// TIA Portal V18 export
DATA_BLOCK "DB 333"   // DB333
{ S7_Optimized_Access := 'FALSE' }
AUTHOR : AWP_S7P
FAMILY : WEB
VERSION : 1.0
// stored: AutoNumber false, DBAccessibleFromOPCUA true, IsOnlyStoredInLoadMemory false, IsWriteProtectedInAS false
   VAR
      magic { ExternalAccessible := 'False'; ExternalVisible := 'False'; ExternalWritable := 'False'} : DWord := DW#16#41575043;
      consistency_tag { ExternalAccessible := 'False'; ExternalVisible := 'False'; ExternalWritable := 'False'} : DWord := DW#16#0F12B01D;
      db_version { ExternalAccessible := 'False'; ExternalVisible := 'False'; ExternalWritable := 'False'} : Word := W#16#0001;
      length { ExternalAccessible := 'False'; ExternalVisible := 'False'; ExternalWritable := 'False'} : UInt := 586;
      pagetab_of { ExternalAccessible := 'False'; ExternalVisible := 'False'; ExternalWritable := 'False'} : UInt := 92;
      pagetab_count { ExternalAccessible := 'False'; ExternalVisible := 'False'; ExternalWritable := 'False'} : UInt := 4;
      excludetab_of { ExternalAccessible := 'False'; ExternalVisible := 'False'; ExternalWritable := 'False'} : UInt := 132;
      excludetab_count { ExternalAccessible := 'False'; ExternalVisible := 'False'; ExternalWritable := 'False'} : UInt := 0;
      fragmentlist_of { ExternalAccessible := 'False'; ExternalVisible := 'False'; ExternalWritable := 'False'} : UInt := 132;
      fragmentlist_count { ExternalAccessible := 'False'; ExternalVisible := 'False'; ExternalWritable := 'False'} : UInt := 5;
      fragmenttab_of { ExternalAccessible := 'False'; ExternalVisible := 'False'; ExternalWritable := 'False'} : UInt := 148;
      fragmenttab_count { ExternalAccessible := 'False'; ExternalVisible := 'False'; ExternalWritable := 'False'} : UInt := 5;
      datatab_of { ExternalAccessible := 'False'; ExternalVisible := 'False'; ExternalWritable := 'False'} : UInt := 218;
      datatab_count { ExternalAccessible := 'False'; ExternalVisible := 'False'; ExternalWritable := 'False'} : UInt := 2;
      usenametab_of { ExternalAccessible := 'False'; ExternalVisible := 'False'; ExternalWritable := 'False'} : UInt := 226;
      usenametab_count { ExternalAccessible := 'False'; ExternalVisible := 'False'; ExternalWritable := 'False'} : UInt := 0;
      enumreftab_of { ExternalAccessible := 'False'; ExternalVisible := 'False'; ExternalWritable := 'False'} : UInt := 226;
      enumreftab_count { ExternalAccessible := 'False'; ExternalVisible := 'False'; ExternalWritable := 'False'} : UInt := 0;
      enumtab_of { ExternalAccessible := 'False'; ExternalVisible := 'False'; ExternalWritable := 'False'} : UInt := 226;
      enumtab_count { ExternalAccessible := 'False'; ExternalVisible := 'False'; ExternalWritable := 'False'} : UInt := 0;
      textlist_of { ExternalAccessible := 'False'; ExternalVisible := 'False'; ExternalWritable := 'False'} : UInt := 226;
      textlist_count { ExternalAccessible := 'False'; ExternalVisible := 'False'; ExternalWritable := 'False'} : UInt := 360;
      language_frag_tab_of { ExternalAccessible := 'False'; ExternalVisible := 'False'; ExternalWritable := 'False'} : UInt := 142;
      language_frag_tab_count { ExternalAccessible := 'False'; ExternalVisible := 'False'; ExternalWritable := 'False'} : UInt := 6;
      application_name { ExternalAccessible := 'False'; ExternalVisible := 'False'; ExternalWritable := 'False'} : UInt := 1;
      application_url { ExternalAccessible := 'False'; ExternalVisible := 'False'; ExternalWritable := 'False'} : UInt := 19;
      application_desc { ExternalAccessible := 'False'; ExternalVisible := 'False'; ExternalWritable := 'False'} : UInt := 29;
      enum_defs_fragment_start { ExternalAccessible := 'False'; ExternalVisible := 'False'; ExternalWritable := 'False'} : UInt := 0;
      enum_defs_fragment_count { ExternalAccessible := 'False'; ExternalVisible := 'False'; ExternalWritable := 'False'} : UInt := 0;
      commandstate { ExternalAccessible := 'False'; ExternalVisible := 'False'; ExternalWritable := 'False'} : Struct
         last_error { ExternalAccessible := 'False'; ExternalVisible := 'False'; ExternalWritable := 'False'} : Int := 0;
         debug_mode { ExternalAccessible := 'False'; ExternalVisible := 'False'; ExternalWritable := 'False'} : Int := 0;
         init { ExternalAccessible := 'False'; ExternalVisible := 'False'; ExternalWritable := 'False'} : Bool := True;
         deactivate { ExternalAccessible := 'False'; ExternalVisible := 'False'; ExternalWritable := 'False'} : Bool := False;
         initializing { ExternalAccessible := 'False'; ExternalVisible := 'False'; ExternalWritable := 'False'} : Bool := False;
         error { ExternalAccessible := 'False'; ExternalVisible := 'False'; ExternalWritable := 'False'} : Bool := False;
         deactivating { ExternalAccessible := 'False'; ExternalVisible := 'False'; ExternalWritable := 'False'} : Bool := False;
         deactivated { ExternalAccessible := 'False'; ExternalVisible := 'False'; ExternalWritable := 'False'} : Bool := False;
         initialized { ExternalAccessible := 'False'; ExternalVisible := 'False'; ExternalWritable := 'False'} : Bool := False;
         reserved1 { ExternalAccessible := 'False'; ExternalVisible := 'False'; ExternalWritable := 'False'} : Bool := False;
         reserved2 { ExternalAccessible := 'False'; ExternalVisible := 'False'; ExternalWritable := 'False'} : Byte := B#16#00;
      END_STRUCT;
      requesttab { ExternalAccessible := 'False'; ExternalVisible := 'False'; ExternalWritable := 'False'} : Array[1..4] of Struct
         page_index { ExternalAccessible := 'False'; ExternalVisible := 'False'; ExternalWritable := 'False'} : UInt;
         fragment_index { ExternalAccessible := 'False'; ExternalVisible := 'False'; ExternalWritable := 'False'} : UInt;
         continue { ExternalAccessible := 'False'; ExternalVisible := 'False'; ExternalWritable := 'False'} : Bool;
         "repeat" { ExternalAccessible := 'False'; ExternalVisible := 'False'; ExternalWritable := 'False'} : Bool;
         abort { ExternalAccessible := 'False'; ExternalVisible := 'False'; ExternalWritable := 'False'} : Bool;
         finish { ExternalAccessible := 'False'; ExternalVisible := 'False'; ExternalWritable := 'False'} : Bool;
         idle { ExternalAccessible := 'False'; ExternalVisible := 'False'; ExternalWritable := 'False'} : Bool;
         waiting { ExternalAccessible := 'False'; ExternalVisible := 'False'; ExternalWritable := 'False'} : Bool;
         sending { ExternalAccessible := 'False'; ExternalVisible := 'False'; ExternalWritable := 'False'} : Bool;
         aborting { ExternalAccessible := 'False'; ExternalVisible := 'False'; ExternalWritable := 'False'} : Bool;
         reserved3 { ExternalAccessible := 'False'; ExternalVisible := 'False'; ExternalWritable := 'False'} : Byte;
      END_STRUCT;
      pagetab { ExternalAccessible := 'False'; ExternalVisible := 'False'; ExternalWritable := 'False'} : Array[1..4] of Struct
         index { ExternalAccessible := 'False'; ExternalVisible := 'False'; ExternalWritable := 'False'} : UInt;
         url { ExternalAccessible := 'False'; ExternalVisible := 'False'; ExternalWritable := 'False'} : UInt;
         mime_type { ExternalAccessible := 'False'; ExternalVisible := 'False'; ExternalWritable := 'False'} : UInt;
         fragment_start { ExternalAccessible := 'False'; ExternalVisible := 'False'; ExternalWritable := 'False'} : UInt;
         fragment_num { ExternalAccessible := 'False'; ExternalVisible := 'False'; ExternalWritable := 'False'} : UInt;
      END_STRUCT;
      fragmentlist { ExternalAccessible := 'False'; ExternalVisible := 'False'; ExternalWritable := 'False'} : Array[1..5] of UInt;
      language_frag_tab { ExternalAccessible := 'False'; ExternalVisible := 'False'; ExternalWritable := 'False'} : Struct
         max_language { ExternalAccessible := 'False'; ExternalVisible := 'False'; ExternalWritable := 'False'} : UInt := 0;
         fragment_count { ExternalAccessible := 'False'; ExternalVisible := 'False'; ExternalWritable := 'False'} : UInt := 0;
         nolang_offset { ExternalAccessible := 'False'; ExternalVisible := 'False'; ExternalWritable := 'False'} : UInt := 0;
      END_STRUCT;
      fragmenttab { ExternalAccessible := 'False'; ExternalVisible := 'False'; ExternalWritable := 'False'} : Array[1..5] of Struct
         fragment_name { ExternalAccessible := 'False'; ExternalVisible := 'False'; ExternalWritable := 'False'} : UInt;
         fragment_type { ExternalAccessible := 'False'; ExternalVisible := 'False'; ExternalWritable := 'False'} : Byte;
         fragment_version { ExternalAccessible := 'False'; ExternalVisible := 'False'; ExternalWritable := 'False'} : Byte;
         content_db { ExternalAccessible := 'False'; ExternalVisible := 'False'; ExternalWritable := 'False'} : UInt;
         content_of { ExternalAccessible := 'False'; ExternalVisible := 'False'; ExternalWritable := 'False'} : UInt;
         content_length { ExternalAccessible := 'False'; ExternalVisible := 'False'; ExternalWritable := 'False'} : UInt;
         data_start { ExternalAccessible := 'False'; ExternalVisible := 'False'; ExternalWritable := 'False'} : UInt;
         data_num { ExternalAccessible := 'False'; ExternalVisible := 'False'; ExternalWritable := 'False'} : UInt;
      END_STRUCT;
      datatab { ExternalAccessible := 'False'; ExternalVisible := 'False'; ExternalWritable := 'False'} : Array[1..2] of Struct
         variable_name { ExternalAccessible := 'False'; ExternalVisible := 'False'; ExternalWritable := 'False'} : UInt;
         direction { ExternalAccessible := 'False'; ExternalVisible := 'False'; ExternalWritable := 'False'} : Int;
      END_STRUCT;
      textlist { ExternalAccessible := 'False'; ExternalVisible := 'False'; ExternalWritable := 'False'} : Array[1..360] of Byte := 434F4E435233444557656253657276657200696E6465782E68746D00434F4E435233444557656253657276657200636F6E63723364655F736F6C6F6C6F676F5F313030783130305F314D335F69636F6E2E69636F006170706C69636174696F6E2F6F637465742D73747265616D00696E6465782E68746D00746578742F68746D6C00494F436F756E7465722E68746D00746578742F68746D6C006A71756572792D322E302E322E6D696E2E6A73006170706C69636174696F6E2F6A61766173637269707400636F6E63723364655F736F6C6F6C6F676F5F313030783130305F314D335F69636F6E2E69636F00696E6465782E68746D00494F436F756E7465722E68746D006A71756572792D322E302E322E6D696E2E6A73006A71756572792D322E302E322E6D696E2E6A735F31002244657654657374426C6F636B222E57656253657276657254657374002244657654657374426C6F636B222E5765625365727665725465737400;
   END_VAR
BEGIN
   requesttab[1..4].page_index := 0;
   requesttab[1..4].fragment_index := 0;
   requesttab[1..4].continue := False;
   requesttab[1..4]."repeat" := False;
   requesttab[1..4].abort := False;
   requesttab[1..4].finish := False;
   requesttab[1..4].idle := False;
   requesttab[1..4].waiting := False;
   requesttab[1..4].sending := False;
   requesttab[1..4].aborting := False;
   requesttab[1..4].reserved3 := B#16#00;
   pagetab[1].index := 1;
   pagetab[2].index := 2;
   pagetab[3].index := 3;
   pagetab[4].index := 4;
   pagetab[1].url := 47;
   pagetab[2].url := 111;
   pagetab[3].url := 131;
   pagetab[4].url := 155;
   pagetab[1].mime_type := 86;
   pagetab[2].mime_type := 121;
   pagetab[3].mime_type := 145;
   pagetab[4].mime_type := 175;
   pagetab[1].fragment_start := 1;
   pagetab[2].fragment_start := 2;
   pagetab[3].fragment_start := 3;
   pagetab[4].fragment_start := 4;
   pagetab[1..3].fragment_num := 1;
   pagetab[4].fragment_num := 2;
   fragmentlist[1] := 1;
   fragmentlist[2] := 2;
   fragmentlist[3] := 3;
   fragmentlist[4] := 4;
   fragmentlist[5] := 5;
   fragmenttab[1].fragment_name := 198;
   fragmenttab[2].fragment_name := 237;
   fragmenttab[3].fragment_name := 247;
   fragmenttab[4].fragment_name := 261;
   fragmenttab[5].fragment_name := 281;
   fragmenttab[1..5].fragment_type := B#16#00;
   fragmenttab[1..5].fragment_version := B#16#00;
   fragmenttab[1..3].content_db := 334;
   fragmenttab[4].content_db := 335;
   fragmenttab[5].content_db := 336;
   fragmenttab[1].content_of := 8;
   fragmenttab[2].content_of := 41248;
   fragmenttab[3].content_of := 42946;
   fragmenttab[4..5].content_of := 8;
   fragmenttab[1].content_length := 41239;
   fragmenttab[2].content_length := 1697;
   fragmenttab[3].content_length := 183;
   fragmenttab[4].content_length := 65526;
   fragmenttab[5].content_length := 17975;
   fragmenttab[1].data_start := 0;
   fragmenttab[2].data_start := 1;
   fragmenttab[3].data_start := 2;
   fragmenttab[4..5].data_start := 0;
   fragmenttab[1].data_num := 0;
   fragmenttab[2..3].data_num := 1;
   fragmenttab[4..5].data_num := 0;
   datatab[1].variable_name := 303;
   datatab[2].variable_name := 332;
   datatab[1..2].direction := 3;
END_DATA_BLOCK
